TYPE ST_DC_Input :
STRUCT
  Input      : BIT;

  Status     : USINT;

  LatchPositive  : ULINT;
  LatchNegative  : ULINT;
END_STRUCT
END_TYPE

(* stored: Version 1.1.0.1
   DUT ST_DC_Input: Id {c3788cae-7d0e-4cb2-8605-55034eab1558} *)
